// TIA Portal V16 export
// export: Created 2023-01-04T15:44:08.6296745Z, ExportSetting WithDefaults, DisplayName Totally Integrated Automation Portal, DisplayVersion V16, DisplayName TIA Portal Version Control Interface, DisplayVersion V16, DisplayName TIA Portal Openness, DisplayVersion V16, DisplayName STEP 7 Professional, DisplayVersion V16, DisplayName STEP 7 Safety, DisplayVersion V16, DisplayName WinCC Advanced, DisplayVersion V16
FUNCTION_BLOCK "Re-filling_Logic"   // FB1, LAD
{ S7_Optimized_Access := 'TRUE' }
VERSION : 0.1
// stored: AutoNumber true, IsIECCheckEnabled false, IsRetainMemResEnabled false, MemoryReserve 100, SetENOAutomatically false, UDAEnableTagReadback false
   VAR_TEMP   // added for the SCL form of the ladder/FBD networks
      _w1 : Bool;
      _w2 : Bool;
      _w3 : Bool;
      _w4 : Bool;
   END_VAR
BEGIN

REGION Network 1: Tank2 Re-filling Proccess
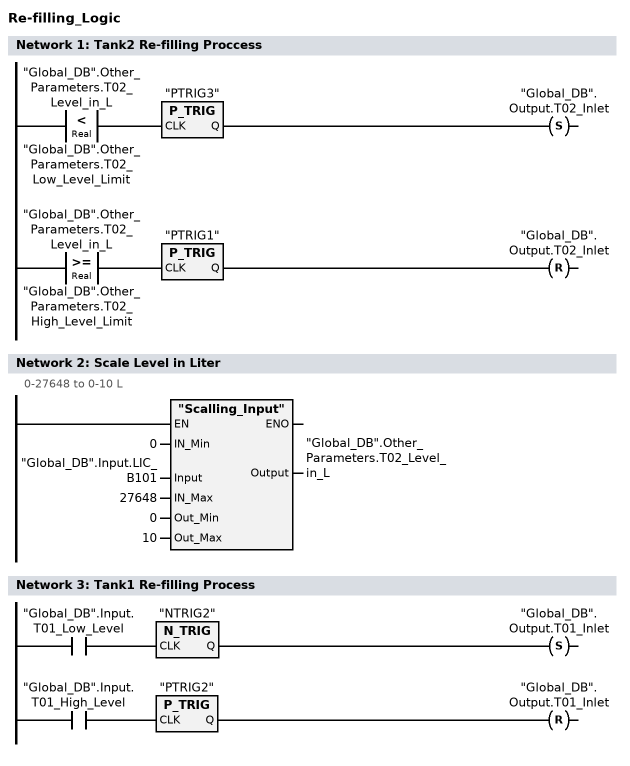
   RUNG wire#powerrail
      { S7_Templates := "SrcType := Real" } LT_Contact(in1 := "Global_DB".Other_Parameters.T02_Level_in_L, in2 := "Global_DB".Other_Parameters.T02_Low_Level_Limit)
      P_Trig( "PTRIG3" )
      S_Coil( "Global_DB".Output.T02_Inlet )
   END_RUNG
   RUNG wire#powerrail
      { S7_Templates := "SrcType := Real" } GE_Contact(in1 := "Global_DB".Other_Parameters.T02_Level_in_L, in2 := "Global_DB".Other_Parameters.T02_High_Level_Limit)
      P_Trig( "PTRIG1" )
      R_Coil( "Global_DB".Output.T02_Inlet )
   END_RUNG
   // the same network as SCL:
   #_w1 := "Global_DB".Other_Parameters.T02_Level_in_L < "Global_DB".Other_Parameters.T02_Low_Level_Limit;
   #_w2 := #_w1 AND NOT "PTRIG3";   // rising edge
   "PTRIG3" := #_w1;
   IF #_w2 THEN "Global_DB".Output.T02_Inlet := TRUE; END_IF;
   #_w3 := "Global_DB".Other_Parameters.T02_Level_in_L >= "Global_DB".Other_Parameters.T02_High_Level_Limit;
   #_w4 := #_w3 AND NOT "PTRIG1";   // rising edge
   "PTRIG1" := #_w3;
   IF #_w4 THEN "Global_DB".Output.T02_Inlet := FALSE; END_IF;
END_REGION

REGION Network 2: Scale Level in Liter
   // 0-27648 to 0-10 L
   RUNG wire#powerrail
      "Scalling_Input"(IN_Min := 0, Input := "Global_DB".Input.LIC_B101, IN_Max := 27648, Out_Min := 0, Out_Max := 10, Output => "Global_DB".Other_Parameters.T02_Level_in_L)
   END_RUNG
   // the same network as SCL:
   "Scalling_Input"(IN_Min := 0,
                    Input := "Global_DB".Input.LIC_B101,
                    IN_Max := 27648,
                    Out_Min := 0,
                    Out_Max := 10,
                    Output => "Global_DB".Other_Parameters.T02_Level_in_L);
END_REGION

REGION Network 3: Tank1 Re-filling Process
   RUNG wire#powerrail
      Contact( "Global_DB".Input.T01_Low_Level )
      N_Trig( "NTRIG2" )
      S_Coil( "Global_DB".Output.T01_Inlet )
   END_RUNG
   RUNG wire#powerrail
      Contact( "Global_DB".Input.T01_High_Level )
      P_Trig( "PTRIG2" )
      R_Coil( "Global_DB".Output.T01_Inlet )
   END_RUNG
   // the same network as SCL:
   #_w1 := NOT "Global_DB".Input.T01_Low_Level AND "NTRIG2";   // falling edge
   "NTRIG2" := "Global_DB".Input.T01_Low_Level;
   IF #_w1 THEN "Global_DB".Output.T01_Inlet := TRUE; END_IF;
   #_w2 := "Global_DB".Input.T01_High_Level AND NOT "PTRIG2";   // rising edge
   "PTRIG2" := "Global_DB".Input.T01_High_Level;
   IF #_w2 THEN "Global_DB".Output.T01_Inlet := FALSE; END_IF;
END_REGION
END_FUNCTION_BLOCK
